(*********************************** G.D S.p.A. - Technical Department ***********************************
============= PROGRAM INFO ============
FOLDER:             TBD
MACHINES INVOLVED:  TBD 

============= DESCRIPTION =============
csp machine declaration

============= REVISIONS ===============
Date		Version	 	Author      	Description             
----------	-------		------------  	--------------------------------------------
2019/04/05 	0000.00	 	M.Grasso		Creation of the PRG

**********************************************************************************************************)
(*$R process_ref := prc; $*)
PROGRAM csp_case_glue_ls
VAR
	
	prc:											process;
	prc_path:										STRING;
	
END_VAR

_read_var_input();

_object_manager();

IF NOT objects_running()
THEN
	RETURN;	
END_IF

_read_process_image();

_mode_manager();

_set_runtime_properties();

(********************************* BODY *********************************)
(************************************************************************)

_handle_messages();

_write_output();

ACTION _handle_messages:
;
END_ACTION

ACTION _handle_process_test:
;
END_ACTION

ACTION _mode_manager:
IF process_mode_req_is_pending(prc)
THEN
    process_apply_mode_req_first_step(prc);
    CASE process_get_mode(prc) OF
        MODE_TO_ABSENT:
			;
        MODE_TO_INACTIVE:
			;
        MODE_TO_TEST:
			;
        MODE_TO_OPERATIONAL:
			;
    END_CASE
    process_apply_mode_req_second_step(prc);
END_IF
END_ACTION

ACTION _object_manager:
IF objects_initialization()
THEN
	sub_process_init(
		object_name					:= 'csp_case_glue_ls.prc', 
		process						:= csp_case_glue.prc, 
		CONVERSION_this				:= prc);
		
	prc_path 						:= process_get_path(prc);
END_IF

IF objects_running()
THEN
	process_cycle(prc);
END_IF
END_ACTION

ACTION _read_process_image:
;
END_ACTION

ACTION _read_var_input:
;
END_ACTION

ACTION _set_runtime_properties:
;
END_ACTION

ACTION _write_output:
;
END_ACTION

END_PROGRAM

(* stored: Version 1.1.0.1, ProductVersion 3.1.4022.12
   POU csp_case_glue_ls: Id {e4d52b73-a097-49ed-bd73-82177cd5c6de}, SpecialFunc None
   Action _handle_messages: Id {9f0010cc-a3ec-4345-a7ba-2de182b14f02}
   Action _handle_process_test: Id {a96e2469-3678-4cf0-8d7d-311bdf3b5521}
   Action _mode_manager: Id {d2b72ba5-d983-4fe8-9018-f3197e81ae82}
   Action _object_manager: Id {8a03bad3-58e0-4b52-8a02-c08b1b1297e7}
   Action _read_process_image: Id {a0c98d76-2441-433a-ada1-566a5ab27e7f}
   Action _read_var_input: Id {5aeaf196-b458-408c-b7b2-4486cc79ba24}
   Action _set_runtime_properties: Id {58d751de-30b6-43f8-a681-bfbd2a9a8c8a}
   Action _write_output: Id {6ce915d9-c656-4255-b31f-f3d1caf9bd2b} *)
